FUNCTION_BLOCK Mc2Halt EXTENDS TaskBase
VAR_INPUT
END_VAR
VAR_OUTPUT
END_VAR
VAR
	mcHalt : Tc2_MC2.MC_Halt;
	_Axis : REFERENCE TO Tc2_MC2.AXIS_REF;
	_Halt : BOOL;
END_VAR

{analysis -2}

METHOD Abort : BOOL
mcHalt.Execute := FALSE;
_Busy := FALSE;
_Halt := FALSE;
Abort := TRUE;
State := 0;
END_METHOD

METHOD Cycle : HRESULT
VAR_INPUT
END_VAR
Cycle := S_OK;
CASE State OF
	0:
		IF _Halt THEN
			Cycle := S_PENDING;
			_Done := FALSE;
			_Error := FALSE;
			_Busy := TRUE;
			mcHalt.Execute := TRUE;
			IF mcHalt.Busy THEN
				State := 10;
				_Halt := FALSE;
			END_IF
		END_IF
	
	10:
		IF NOT mcHalt.Busy THEN
			IF mcHalt.Done THEN
				_Done := TRUE;
			ELSIF mcHalt.Error THEN
				_Error := TRUE;
			END_IF
			_Busy := FALSE;
			mcHalt.Execute := FALSE;
			State := 0;
			Cycle := S_OK;
		END_IF
	ELSE
		Cycle := E_FAIL;
END_CASE

mcHalt(Axis := _Axis);
END_METHOD

METHOD Execute : HRESULT
VAR_INPUT
END_VAR
IF _Axis.Status.Moving THEN
	Execute := S_OK;
	_Halt := TRUE;
END_IF
END_METHOD

METHOD FB_init : BOOL
VAR_INPUT
	bInitRetains : BOOL; // if TRUE, the retain variables are initialized (warm start / cold start)
	bInCopyCode : BOOL;  // if TRUE, the instance afterwards gets moved into the copy code (online change)
	axis : reference TO AXIS_REF;
END_VAR
_Axis REF= axis;
END_METHOD

END_FUNCTION_BLOCK

(* stored: Version 1.1.0.1
   POU Mc2Halt: Id {8f902aee-94bf-4385-bdcf-ca790f894752}, SpecialFunc None
   Method Abort: Id {628339b1-4bd1-432e-8277-d60f3e75db0d}
   Method Cycle: Id {82fe1e7b-ab2b-4a89-9b59-5eb25d835959}
   Method Execute: Id {020a5dad-2d55-4c66-8489-dc08945209ce}
   Method FB_init: Id {1d755e0d-6917-492a-87c8-d14e7bb31076} *)
